FUNCTION F_SettingItemHandlingF : LREAL
VAR_IN_OUT
	fValue 		: LREAL;
	stSetting 	: ST_Data_Item;
END_VAR
VAR
	stInfo 		: ST_Text;
	sChanges	: T_MaxString;
	IEvent		: I_EventHandler;
END_VAR

F_SettingItemHandlingF := stSetting.fValue;

IF Services.bSettingsSaved OR NOT Services.bPlcInitDone THEN
	fValue := stSetting.fValue;
	RETURN;
END_IF

IF ABS(fValue - stSetting.fValue) < Statics.fEpsilon THEN
	RETURN;
END_IF

sChanges := sEmpty;
IEvent := Services.fbEventHandler;

// 1. chk user level
IF NOT F_ChkSettingUserLevel(HMI.eUserLevel, stSetting, stInfo => stInfo) THEN							  
	IEvent.Select(TC_Events.SettingsEventClass.WarningEvent)
		  .ArgAddWString(stInfo.wsName)
		  .Raise();
							
	fValue := stSetting.fValue;
	RETURN;
END_IF


// 2. chk min/max value
IF NOT F_ChkSettingLimitF(fValue, stSetting, stInfo => stInfo) THEN
	IEvent.Select(TC_Events.SettingsEventClass.WarningEvent)
		  .ArgAddWString(stInfo.wsName)
		  .Raise();
							
	fValue := stSetting.fValue;
	RETURN;
END_IF

// 3. save changes
IF stSetting.eDataType = E_DataType.eDataType_bool THEN
	F_TrackSettingChangesB(fValue = 1, stSetting, sChanges);
ELSIF stSetting.eDataType = E_DataType.eDataType_int THEN
	F_TrackSettingChangesI(TO_INT(fValue), stSetting, sChanges);
ELSIF stSetting.eDataType = E_DataType.eDataType_lreal THEN
	F_TrackSettingChangesF(fValue, stSetting, sChanges);
ELSIF stSetting.eDataType = E_DataType.eDataType_wstring THEN
	F_TrackSettingChangesWs(TO_WSTRING(fValue), stSetting, sChanges);
ELSIF stSetting.eDataType = E_DataType.eDataType_time_ms THEN
	F_TrackSettingChangesT(TO_TIME(fValue), stSetting, sChanges);
ELSIF stSetting.eDataType = E_DataType.eDataType_time_s THEN
	F_TrackSettingChangesT(TO_TIME(fValue * 1000), stSetting, sChanges);
ELSIF stSetting.eDataType = E_DataType.eDataType_time_m THEN
	F_TrackSettingChangesT(TO_TIME(fValue * 60000), stSetting, sChanges);
ELSIF stSetting.eDataType = E_DataType.eDataType_time_h THEN
	F_TrackSettingChangesT(TO_TIME(fValue * 360000),stSetting, sChanges);
END_IF

// 4. track settings changes
IF sChanges <> sEmpty THEN
	ILog.AddLog(Concat5('Settings Changed, ', 'EKS level: ', TO_STRING(HMI.eUserLevel), '. Changes: ', sChanges), 
				'HMI Controller', 
				E_LogLevel.eLogLevel_info);
END_IF

fValue := stSetting.fValue;
F_SettingItemHandlingF := stSetting.fValue;

END_FUNCTION

(* stored: Version 1.1.0.1
   POU F_SettingItemHandlingF: Id {8703c33f-f273-42d4-a4ff-4d49365418d7}, SpecialFunc None *)
